// TwinCAT 3 PLC project ProjectC
// ProgramVersion: 3.1.4022.7
// libraries:
//   SampleLibraryA, * (blark-testing)
//   Tc2_Standard, * (Beckhoff Automation GmbH)
//   Tc2_System, * (Beckhoff Automation GmbH)
//   Tc3_Module, * (Beckhoff Automation GmbH)
// project tree:
//   / PlcTask.TcTTO
//   POUs/ MAIN.TcPOU
// real-time tasks:
//   TASK PlcTask: cycle T#10ms, priority 20, ADS port 350
// motion (NC):

CONFIGURATION ProjectC
    RESOURCE PLC ON TwinCAT3
        TASK PlcTask(INTERVAL := T#10ms, PRIORITY := 20);
        PROGRAM MAIN WITH PlcTask : MAIN;
    END_RESOURCE
END_CONFIGURATION

// ---- POUs/MAIN.TcPOU
PROGRAM MAIN
VAR
	{attribute 'pytmc' := 'pv: PREFIX:fbTest'}
	fbTest : FB_SampleA_Test;
	{attribute 'pytmc' := 'pv: PREFIX:fOutput'}
	fOutput : LREAL;
END_VAR

fbTest(fInput:=1.0, fOutput=>fOutput);

END_PROGRAM
